PROGRAM MAIN
VAR
	bStartStop: BOOL := FALSE;
	bPulse: BOOL := FALSE;
	
	fbSWG : FB_SquareWaveGenerator;
END_VAR
VAR CONSTANT
	HIGHTIME : TIME := T#2S;
	LOWTIME : TIME := T#3S;
END_VAR

fbSWG(
	bStartStop := bStartStop, 
	tHighTime := HIGHTIME,
	tLowTime := LOWTIME,
	bOutPulse => bPulse);

END_PROGRAM

(* stored: Version 1.1.0.1, ProductVersion 3.1.4024.12
   POU MAIN: Id {de9791fb-a451-4f8e-9bb5-6b40ceb12777}, SpecialFunc None *)
